TYPE EN_SequenceState :
(
	SequenceStateActive := 0,
	SequenceStateError,
	SequenceStateWaiting,
	SequenceStateHalt,
	SequenceStateStop,
	SequenceStateInit,
	SequenceStateStep
);
END_TYPE

(* stored: Version 1.1.0.1, ProductVersion 3.1.0.36
   DUT EN_SequenceState: Id {4a76a724-a416-42d9-ba02-afcd4be10203} *)
